{attribute addProperty BoxType "EL9576-0000-0019"}
{attribute addProperty Id "BCT_InputsAT %I*BCT_Inputs_6A3D8194136170WcStateAT %I*WcState_98A4DF7520.250InfoDataAT %I*InfoData_BC63D37F80100"}
{attribute addProperty CRC "66584641"}
{attribute addProperty SizeInBites "218"}
{attribute addProperty SizeInBytes "27.25"}
TYPE EL9576_8602C5C4 :
STRUCT
	{attribute addProperty Name "BCT_Inputs"}
	BCT_Inputs : BCT_Inputs_6A3D8194;
	{attribute addProperty Name "WcState"}
	WcState : WcState_98A4DF75;
	{attribute addProperty Name "InfoData"}
	InfoData : InfoData_BC63D37F;
END_STRUCT
END_TYPE

(* stored: Version 1.2.0.0, ProductVersion 3.1.4024.9
   DUT EL9576_8602C5C4: Id {4f08f44a-19fb-4cd4-b5ab-a3da639b81b7} *)
